// TIA Portal V20 export
VAR_GLOBAL   // PLC tag table "LGR_Const_Measure"
END_VAR
VAR_GLOBAL CONSTANT   // user constants
   MEAS_STAT_NONE : UInt := 0;   // Measure status: none / initial / 측정 상태: 없음(초기)
   MEAS_STAT_BUSY : UInt := 1;   // Measure status: measuring / 측정 상태: 측정 중
   MEAS_STAT_DONE : UInt := 2;   // Measure status: done / 측정 상태: 완료
   MEAS_STAT_ERROR : UInt := 3;   // Measure status: error / 측정 상태: 실패
   MEAS_STAT_MISMATCH : UInt := 4;   // Measure status: done but laser/torque inner dia mismatch / 측정 상태: 완료(레이저/토크 내경 불일치)
   MEAS_STAT_SKU_COUNT_MISMATCH : UInt := 5;   // SKU done - stack count differs by direction (X0) / SKU 완료 - 방향별 단수 불일치 (DiagFlags X0)
   MEAS_STAT_SKU_HEIGHT_SPREAD : UInt := 6;   // SKU done - exit height spread over limit (X1) / SKU 완료 - 방향별 이탈 높이 편차 초과 (DiagFlags X1)
   MEAS_STAT_SKU_LAYER_OFFSET : UInt := 7;   // SKU done - layer center offset over limit (X4) / SKU 완료 - 단별 편심 초과, 삐뚤게 쌓임 (DiagFlags X4)
   MEAS_STAT_SKU_LIFT_END : UInt := 8;   // SKU done - finished at lift end before all exits (X6) / SKU 완료 - 모두 빠져나가기 전 리프트 끝 확정 (DiagFlags X6)
   MEAS_STAT_SKU_NO_EDGE : UInt := 9;   // SKU done - no exit edge (X7) / SKU 완료 - 이탈 경계 없음 (DiagFlags X7)
   MEAS_STAT_SKU_CMD_COUNT : UInt := 10;   // SKU done - measured stack count differs from commanded Item.Count (X8, error) / SKU 완료 - 상위 명령 단수와 측정 단수 불일치 (DiagFlags X8, 오류)
   MEAS_SKU_STATUS : Int := 0;   // SKU.Data index: status (MEAS_STAT_*) / SKU.Data 인덱스: 상태
   MEAS_SKU_STACK1_LOWER : Int := 1;   // SKU.Data index: stack #1 lower bead pos / SKU.Data 인덱스: 1단 하비드
   MEAS_SKU_STACK1_UPPER : Int := 2;   // SKU.Data index: stack #1 upper bead pos / SKU.Data 인덱스: 1단 상비드
   MEAS_SKU_STACK2_LOWER : Int := 3;   // SKU.Data index: stack #2 lower bead pos / SKU.Data 인덱스: 2단 하비드
   MEAS_SKU_STACK2_UPPER : Int := 4;   // SKU.Data index: stack #2 upper bead pos / SKU.Data 인덱스: 2단 상비드
   MEAS_SKU_STACK3_LOWER : Int := 5;   // SKU.Data index: stack #3 lower bead pos / SKU.Data 인덱스: 3단 하비드
   MEAS_SKU_STACK3_UPPER : Int := 6;   // SKU.Data index: stack #3 upper bead pos / SKU.Data 인덱스: 3단 상비드
   MEAS_SKU_STACK4_LOWER : Int := 7;   // SKU.Data index: stack #4 lower bead pos / SKU.Data 인덱스: 4단 하비드
   MEAS_SKU_STACK4_UPPER : Int := 8;   // SKU.Data index: stack #4 upper bead pos / SKU.Data 인덱스: 4단 상비드
   MEAS_SKU_STACK5_LOWER : Int := 9;   // SKU.Data index: stack #5 lower bead pos / SKU.Data 인덱스: 5단 하비드
   MEAS_SKU_STACK5_UPPER : Int := 10;   // SKU.Data index: stack #5 upper bead pos / SKU.Data 인덱스: 5단 상비드
   MEAS_SKU_STACK6_LOWER : Int := 11;   // SKU.Data index: stack #6 lower bead pos / SKU.Data 인덱스: 6단 하비드
   MEAS_SKU_STACK6_UPPER : Int := 12;   // SKU.Data index: stack #6 upper bead pos / SKU.Data 인덱스: 6단 상비드
   MEAS_SKU_STACK7_LOWER : Int := 13;   // SKU.Data index: stack #7 lower bead pos / SKU.Data 인덱스: 7단 하비드
   MEAS_SKU_STACK7_UPPER : Int := 14;   // SKU.Data index: stack #7 upper bead pos / SKU.Data 인덱스: 7단 상비드
   MEAS_SKU_DIAG_FLAGS : Int := 15;   // SKU stack alignment diag flags (FUNC.MeasureSku.DiagFlags as word value) / SKU 스택 정렬 진단 플래그 (FUNC.MeasureSku.DiagFlags, Word 값)
   MEAS_SKU_LAYER_OFFSET : Int := 16;   // SKU max layer center offset (mm) / SKU 단별 편심 최대 (mm)
   MEAS_SKU_TOTAL_COUNT : Int := 17;   // SKU.Data index: stack total count / SKU.Data 인덱스: 스택 단수
   MEAS_SKU_EACH_HEIGHT : Int := 18;   // SKU.Data index: top tire height / SKU.Data 인덱스: 최상단 타이어 높이
   MEAS_SKU_TOTAL_HEIGHT : Int := 19;   // SKU.Data index: stack total height / SKU.Data 인덱스: 스택 전체 높이
   MEAS_ITEM_STATUS : Int := 0;   // Item.Data [COMMON] status / Item.Data [공통] 상태
   MEAS_ITEM_INNER_DIA : Int := 1;   // Item.Data [COMMON] inner diameter (laser in/out vs torque reconciled) / Item.Data [공통] 내경(정합)
   MEAS_ITEM_UPPER_BEAD_HEIGHT : Int := 2;   // Item.Data [COMMON] upper bead height (in/out average) / Item.Data [공통] 상단 비드 높이
   MEAS_ITEM_TIRE_HEIGHT : Int := 3;   // Item.Data [COMMON] tire height (in/out average) / Item.Data [공통] 타이어 높이
   MEAS_ITEM_TORQ_INNER_DIA : Int := 7;   // Item.Data [TORQ] inner diameter by torque grip (avg - 5 mm) / Item.Data [토크] 토크 내경(보정 평균)
   MEAS_ITEM_TORQ_FACTOR : Int := 8;   // Item.Data [TORQ] torque limit factor used / Item.Data [토크] 토크 계수
   MEAS_ITEM_IN_INNER_DIA : Int := 10;   // Item.Data [IN] inner diameter (laser circle fit on insertion) / Item.Data [들어갈 때] 내경
   MEAS_ITEM_IN_UPPER_BEAD_HEIGHT : Int := 11;   // Item.Data [IN] upper bead height (laser closest Z) / Item.Data [들어갈 때] 상단 비드 높이
   MEAS_ITEM_IN_TIRE_HEIGHT : Int := 12;   // Item.Data [IN] tire height (outside->inside edge Z) / Item.Data [들어갈 때] 타이어 높이
   MEAS_ITEM_IN_OFFSET_X : Int := 13;   // Item.Data [IN] centre offset X / Item.Data [들어갈 때] 편심 X
   MEAS_ITEM_IN_OFFSET_Y : Int := 14;   // Item.Data [IN] centre offset Y / Item.Data [들어갈 때] 편심 Y
   MEAS_ITEM_OUT_INNER_DIA : Int := 15;   // Item.Data [OUT] inner diameter (laser circle fit on lift-out) / Item.Data [나갈 때] 내경
   MEAS_ITEM_OUT_UPPER_BEAD_HEIGHT : Int := 16;   // Item.Data [OUT] upper bead height (laser closest Z) / Item.Data [나갈 때] 상단 비드 높이
   MEAS_ITEM_OUT_TIRE_HEIGHT : Int := 17;   // Item.Data [OUT] tire height (inside->outside edge Z) / Item.Data [나갈 때] 타이어 높이
   MEAS_ITEM_OUT_OFFSET_X : Int := 18;   // Item.Data [OUT] centre offset X / Item.Data [나갈 때] 편심 X
   MEAS_ITEM_OUT_OFFSET_Y : Int := 19;   // Item.Data [OUT] centre offset Y / Item.Data [나갈 때] 편심 Y
   MEAS_LOG_ITEM : USInt := 1;   // 측정 이력 종류 : MeasureItem (MEASLOG.Last/Stat 인덱스)
   MEAS_LOG_SKU : USInt := 2;   // 측정 이력 종류 : MeasureSku
   MEAS_LOG_FLOOR : USInt := 3;   // 측정 이력 종류 : MeasureFloor
   MEAS_LOG_PICK : USInt := 4;   // 측정 이력 종류 : PICK 하강 마지막 비드 측정
   MEAS_LOG_MANUAL : USInt := 5;   // 측정 이력 종류 : 수동 측정 (PL_ManualMeasureItem)
   MEAS_LOG_LAST : Int := 199;   // 측정 이력 링버퍼 마지막 인덱스 (MEASLOG.Entry[0..199])
   MEAS_LOG_CODE_LAST : Int := 31;   // 동일 규격(Item Code) 별 누적 슬롯 마지막 인덱스 (MEASLOG.ByCode[0..31])
END_VAR
